FUNCTION_BLOCK Tiempo_TIME_to_seg
VAR_INPUT
	tTime:TIME;
END_VAR
VAR_OUTPUT
	Segundos:DINT;
END_VAR
VAR
END_VAR

Segundos:=TIME_TO_DINT (tTime)/100;

END_FUNCTION_BLOCK

(* stored: Version 1.1.0.1, ProductVersion 3.1.4024.12
   POU Tiempo_TIME_to_seg: Id {b55aca34-9aec-4226-a732-36ff13841020}, SpecialFunc None *)
